# EPICS substitutions: db/Beckhoff_4XXX/ecmcEL4732_s1.substitutions
file "ecmcEcSlave.template"
{
  pattern {}
          {}
}

file "ecmcEL47XX-chX.template"
{
  pattern {CH_ID, DTYP,              FTVL,  NELM}
          {1,     asynInt16ArrayOut, SHORT, 1  }
          {2,     asynInt16ArrayOut, SHORT, 1  }
}
